PROGRAM MBUS_WZaehler2 (* hier wird die Klemme, an welche der M-Bus mit den Zählern angeschlossen ist, alle 10ms aufgerufen *)
VAR
	Komm_Klemme_WZaehler2		: FB_MBUSKL6781;
	WMZ135						: FB_MBUS_General_Ext;
	WMZ138						: FB_MBUS_General_Ext;
	WMZ105						: FB_MBUS_General_Ext;
	WMZ710						: FB_MBUS_General_Ext;
	WMZ205						: FB_MBUS_General_Ext;
	WMZ720						: FB_MBUS_General_Ext;

	adrWMZ135			: ST_MBus_SecAdr := (udiIdNumber:=16#13859504);
	adrWMZ138			: ST_MBus_SecAdr := (udiIdNumber:=16#13859500);
	adrWMZ105			: ST_MBus_SecAdr := (udiIdNumber:=16#12675097);
	adrWMZ205			: ST_MBus_SecAdr := (udiIdNumber:=16#13859501);
	adrWMZ710			: ST_MBus_SecAdr := (udiIdNumber:=16#12675093);
	adrWMZ720			: ST_MBus_SecAdr := (udiIdNumber:=16#13859505);
	
	fbcatch2 : 	Error_Catch;
END_VAR

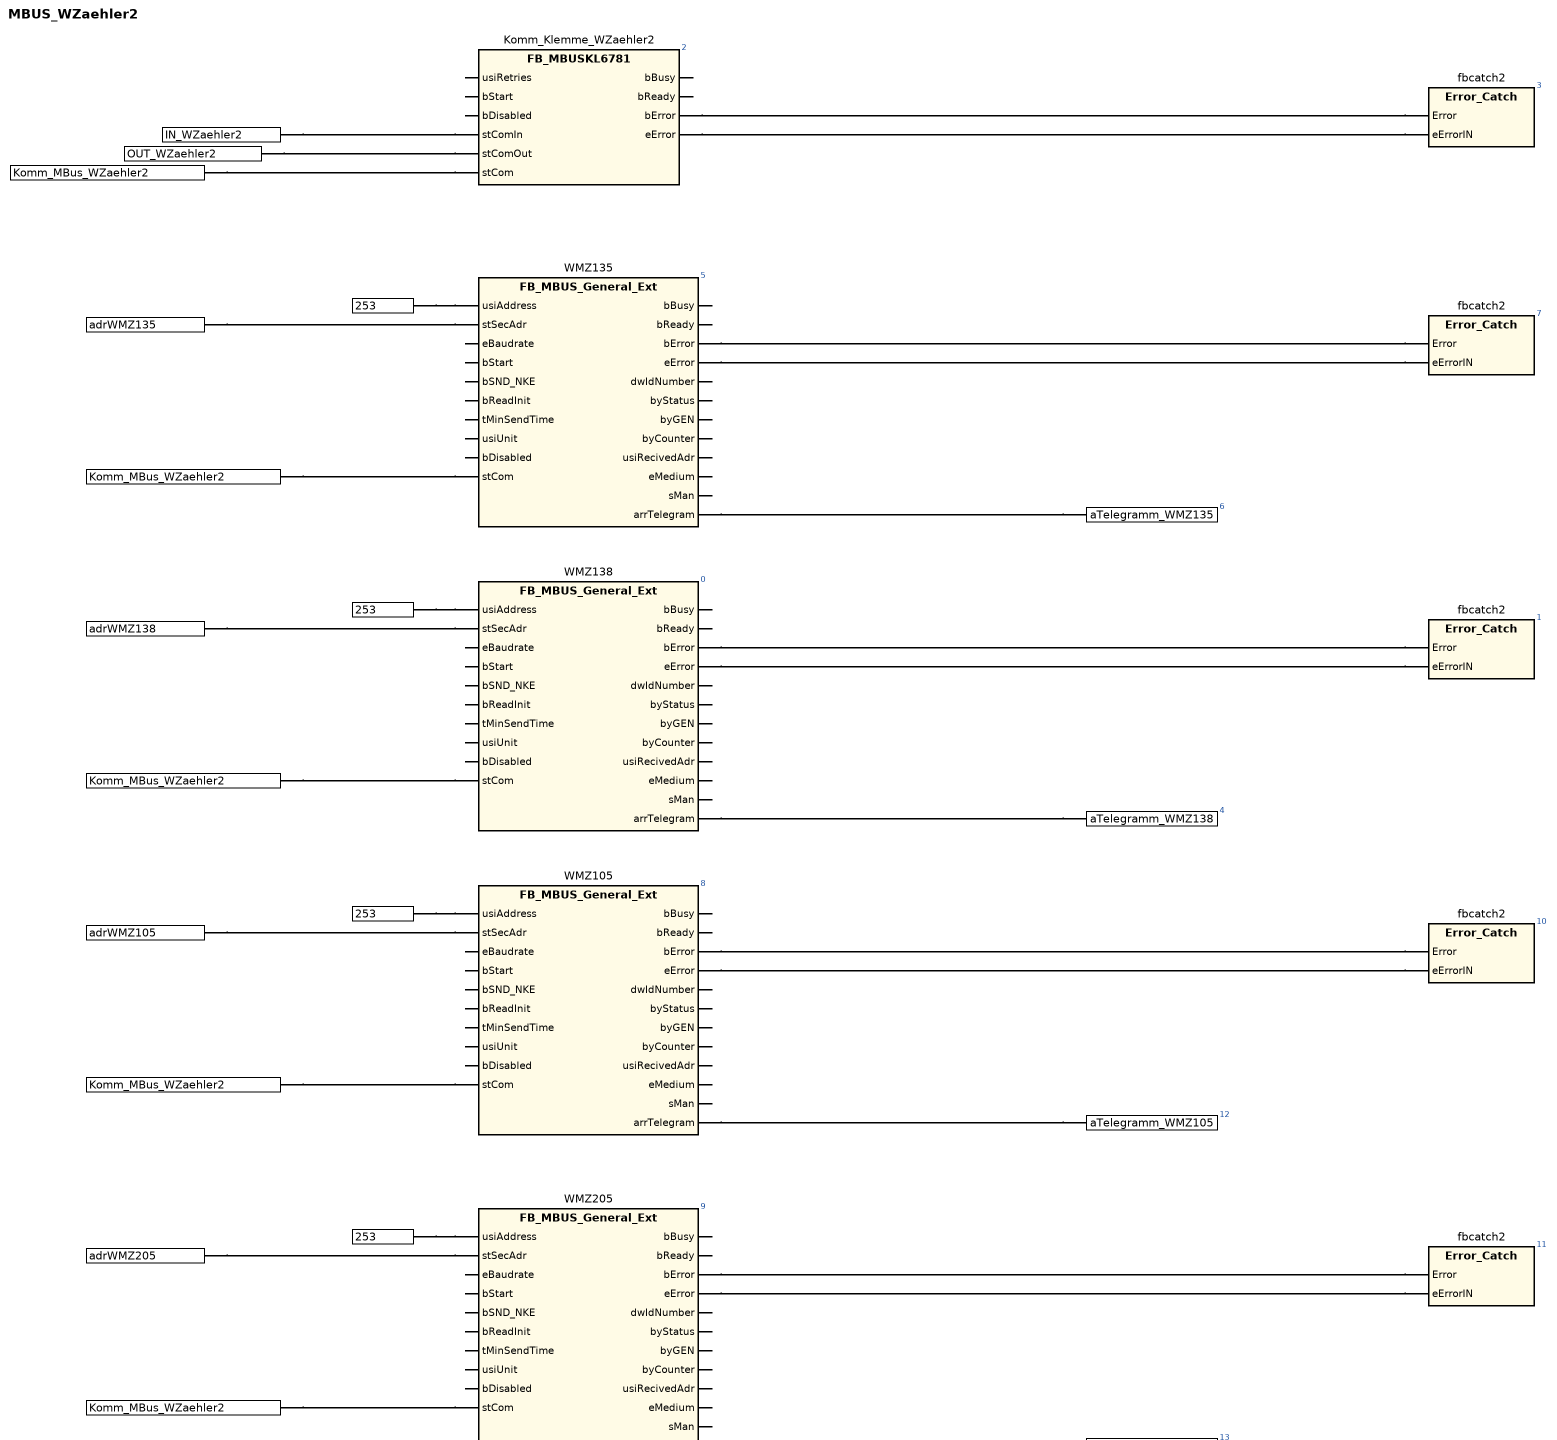
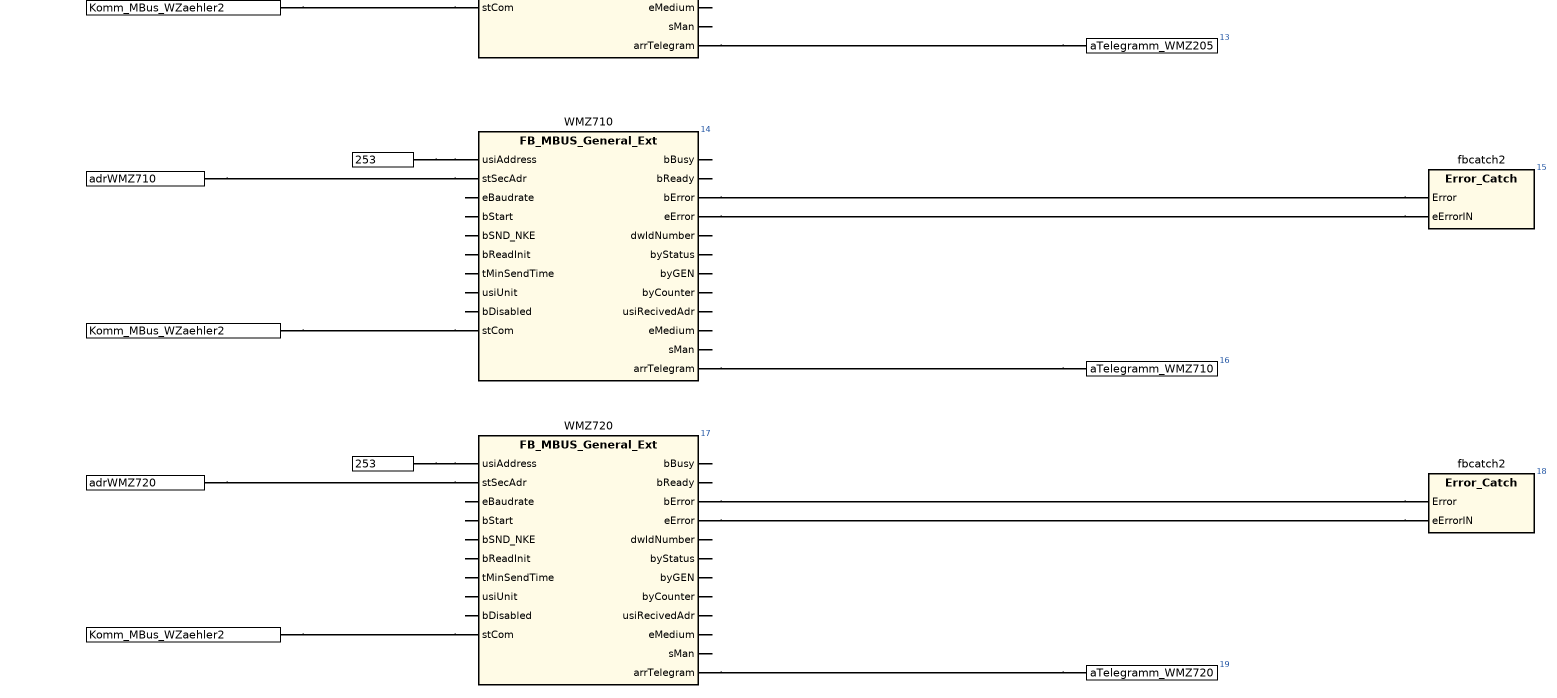
WMZ138(usiAddress := 253, stSecAdr := adrWMZ138, stCom := Komm_MBus_WZaehler2); // FB_MBUS_General_Ext
fbcatch2(Error := WMZ138.bError, eErrorIN := WMZ138.eError); // Error_Catch
Komm_Klemme_WZaehler2(stComIn := IN_WZaehler2, stComOut := OUT_WZaehler2, stCom := Komm_MBus_WZaehler2); // FB_MBUSKL6781
fbcatch2(Error := Komm_Klemme_WZaehler2.bError, eErrorIN := Komm_Klemme_WZaehler2.eError); // Error_Catch
aTelegramm_WMZ138 := WMZ138.arrTelegram;
WMZ135(usiAddress := 253, stSecAdr := adrWMZ135, stCom := Komm_MBus_WZaehler2); // FB_MBUS_General_Ext
aTelegramm_WMZ135 := WMZ135.arrTelegram;
fbcatch2(Error := WMZ135.bError, eErrorIN := WMZ135.eError); // Error_Catch
WMZ105(usiAddress := 253, stSecAdr := adrWMZ105, stCom := Komm_MBus_WZaehler2); // FB_MBUS_General_Ext
WMZ205(usiAddress := 253, stSecAdr := adrWMZ205, stCom := Komm_MBus_WZaehler2); // FB_MBUS_General_Ext
fbcatch2(Error := WMZ105.bError, eErrorIN := WMZ105.eError); // Error_Catch
fbcatch2(Error := WMZ205.bError, eErrorIN := WMZ205.eError); // Error_Catch
aTelegramm_WMZ105 := WMZ105.arrTelegram;
aTelegramm_WMZ205 := WMZ205.arrTelegram;
WMZ710(usiAddress := 253, stSecAdr := adrWMZ710, stCom := Komm_MBus_WZaehler2); // FB_MBUS_General_Ext
fbcatch2(Error := WMZ710.bError, eErrorIN := WMZ710.eError); // Error_Catch
aTelegramm_WMZ710 := WMZ710.arrTelegram;
WMZ720(usiAddress := 253, stSecAdr := adrWMZ720, stCom := Komm_MBus_WZaehler2); // FB_MBUS_General_Ext
fbcatch2(Error := WMZ720.bError, eErrorIN := WMZ720.eError); // Error_Catch
aTelegramm_WMZ720 := WMZ720.arrTelegram;

END_PROGRAM

(* stored: Version 1.1.0.1, ProductVersion 3.1.4024.10
   POU MBUS_WZaehler2: Id {3a3b2554-4e7f-4917-b848-a0dd88abd28f}, SpecialFunc None *)
